PROGRAM Y_Axis
VAR

END_VAR



TrucY();

METHOD TrucY : BOOL
VAR_INPUT
END_VAR
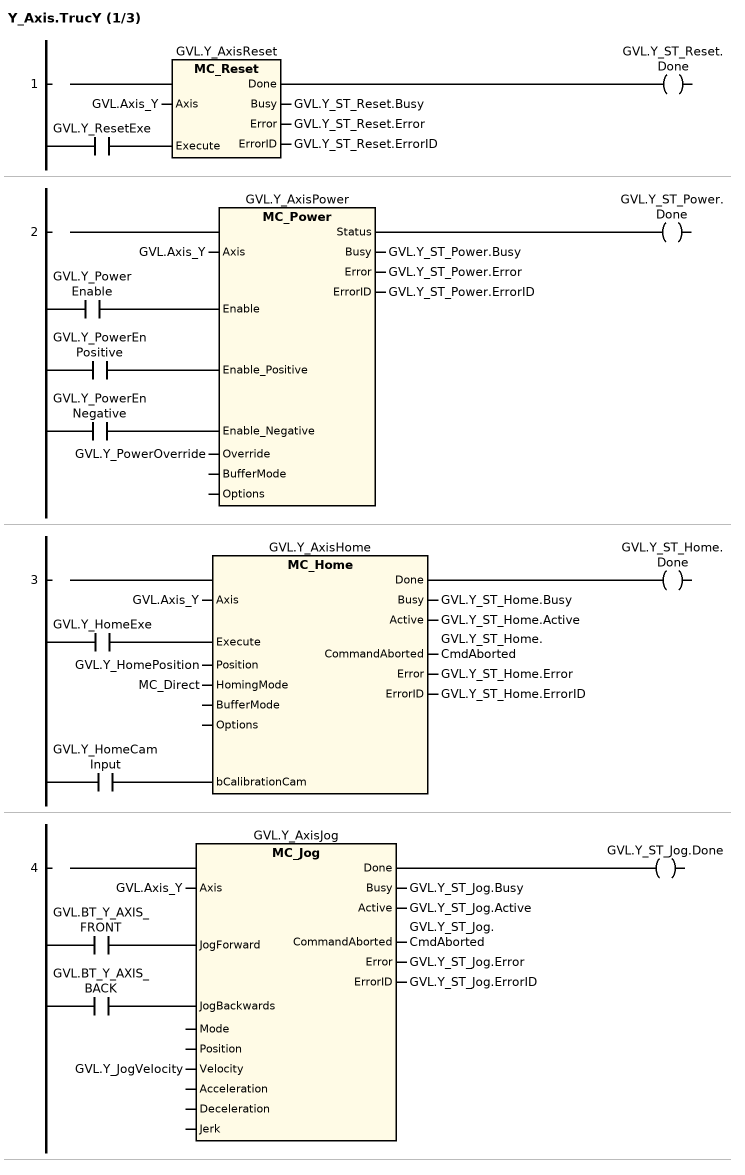
// NETWORK 1
GVL.Y_AxisReset(
    Axis := GVL.Axis_Y,
    Execute := GVL.Y_ResetExe,
    Busy => GVL.Y_ST_Reset.Busy,
    Error => GVL.Y_ST_Reset.Error,
    ErrorID => GVL.Y_ST_Reset.ErrorID); // MC_Reset
GVL.Y_ST_Reset.Done := GVL.Y_AxisReset.Done;

// NETWORK 2
GVL.Y_AxisPower(
    Axis := GVL.Axis_Y,
    Enable := GVL.Y_PowerEnable,
    Enable_Positive := GVL.Y_PowerEnPositive,
    Enable_Negative := GVL.Y_PowerEnNegative,
    Override := GVL.Y_PowerOverride,
    Busy => GVL.Y_ST_Power.Busy,
    Error => GVL.Y_ST_Power.Error,
    ErrorID => GVL.Y_ST_Power.ErrorID); // MC_Power
GVL.Y_ST_Power.Done := GVL.Y_AxisPower.Status;

// NETWORK 3
GVL.Y_AxisHome(
    Axis := GVL.Axis_Y,
    Execute := GVL.Y_HomeExe,
    Position := GVL.Y_HomePosition,
    HomingMode := MC_Direct,
    bCalibrationCam := GVL.Y_HomeCamInput,
    Busy => GVL.Y_ST_Home.Busy,
    Active => GVL.Y_ST_Home.Active,
    CommandAborted => GVL.Y_ST_Home.CmdAborted,
    Error => GVL.Y_ST_Home.Error,
    ErrorID => GVL.Y_ST_Home.ErrorID); // MC_Home
GVL.Y_ST_Home.Done := GVL.Y_AxisHome.Done;

// NETWORK 4
GVL.Y_AxisJog(
    Axis := GVL.Axis_Y,
    JogForward := GVL.BT_Y_AXIS_FRONT,
    JogBackwards := GVL.BT_Y_AXIS_BACK,
    Velocity := GVL.Y_JogVelocity,
    Busy => GVL.Y_ST_Jog.Busy,
    Active => GVL.Y_ST_Jog.Active,
    CommandAborted => GVL.Y_ST_Jog.CmdAborted,
    Error => GVL.Y_ST_Jog.Error,
    ErrorID => GVL.Y_ST_Jog.ErrorID); // MC_Jog
GVL.Y_ST_Jog.Done := GVL.Y_AxisJog.Done;

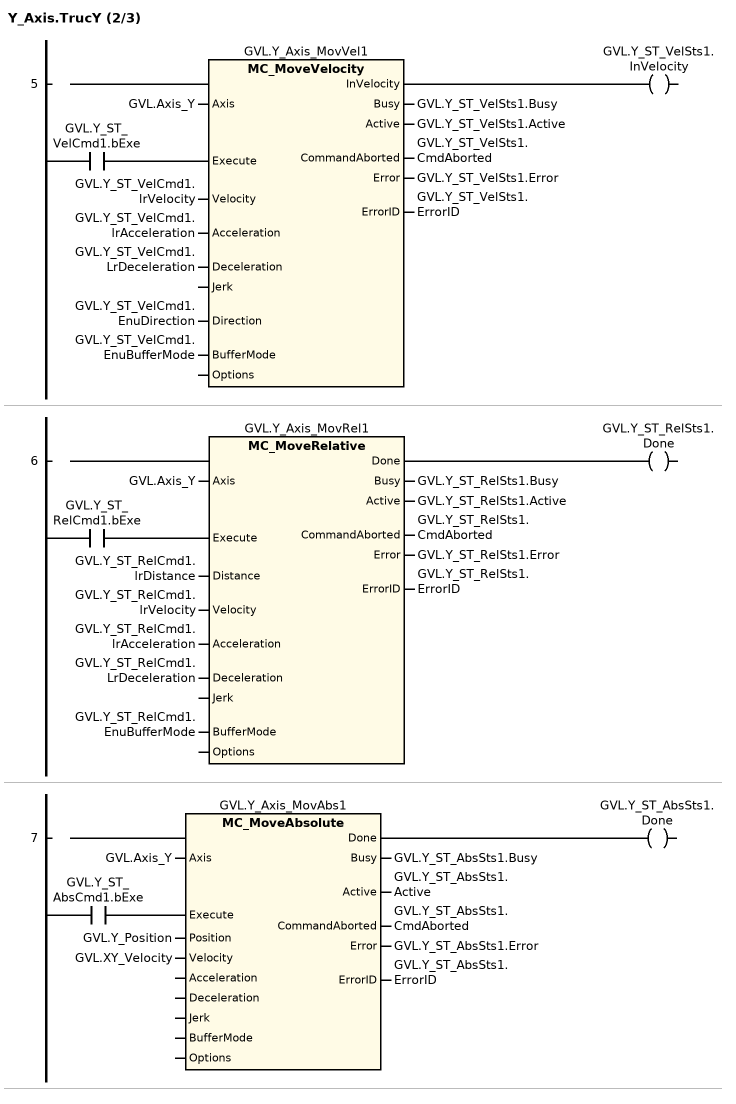
// NETWORK 5
GVL.Y_Axis_MovVel1(
    Axis := GVL.Axis_Y,
    Execute := GVL.Y_ST_VelCmd1.bExe,
    Velocity := GVL.Y_ST_VelCmd1.lrVelocity,
    Acceleration := GVL.Y_ST_VelCmd1.lrAcceleration,
    Deceleration := GVL.Y_ST_VelCmd1.LrDeceleration,
    Direction := GVL.Y_ST_VelCmd1.EnuDirection,
    BufferMode := GVL.Y_ST_VelCmd1.EnuBufferMode,
    Busy => GVL.Y_ST_VelSts1.Busy,
    Active => GVL.Y_ST_VelSts1.Active,
    CommandAborted => GVL.Y_ST_VelSts1.CmdAborted,
    Error => GVL.Y_ST_VelSts1.Error,
    ErrorID => GVL.Y_ST_VelSts1.ErrorID); // MC_MoveVelocity
GVL.Y_ST_VelSts1.InVelocity := GVL.Y_Axis_MovVel1.InVelocity;

// NETWORK 6
GVL.Y_Axis_MovRel1(
    Axis := GVL.Axis_Y,
    Execute := GVL.Y_ST_RelCmd1.bExe,
    Distance := GVL.Y_ST_RelCmd1.lrDistance,
    Velocity := GVL.Y_ST_RelCmd1.lrVelocity,
    Acceleration := GVL.Y_ST_RelCmd1.lrAcceleration,
    Deceleration := GVL.Y_ST_RelCmd1.LrDeceleration,
    BufferMode := GVL.Y_ST_RelCmd1.EnuBufferMode,
    Busy => GVL.Y_ST_RelSts1.Busy,
    Active => GVL.Y_ST_RelSts1.Active,
    CommandAborted => GVL.Y_ST_RelSts1.CmdAborted,
    Error => GVL.Y_ST_RelSts1.Error,
    ErrorID => GVL.Y_ST_RelSts1.ErrorID); // MC_MoveRelative
GVL.Y_ST_RelSts1.Done := GVL.Y_Axis_MovRel1.Done;

// NETWORK 7
GVL.Y_Axis_MovAbs1(
    Axis := GVL.Axis_Y,
    Execute := GVL.Y_ST_AbsCmd1.bExe,
    Position := GVL.Y_Position,
    Velocity := GVL.XY_Velocity,
    Busy => GVL.Y_ST_AbsSts1.Busy,
    Active => GVL.Y_ST_AbsSts1.Active,
    CommandAborted => GVL.Y_ST_AbsSts1.CmdAborted,
    Error => GVL.Y_ST_AbsSts1.Error,
    ErrorID => GVL.Y_ST_AbsSts1.ErrorID); // MC_MoveAbsolute
GVL.Y_ST_AbsSts1.Done := GVL.Y_Axis_MovAbs1.Done;

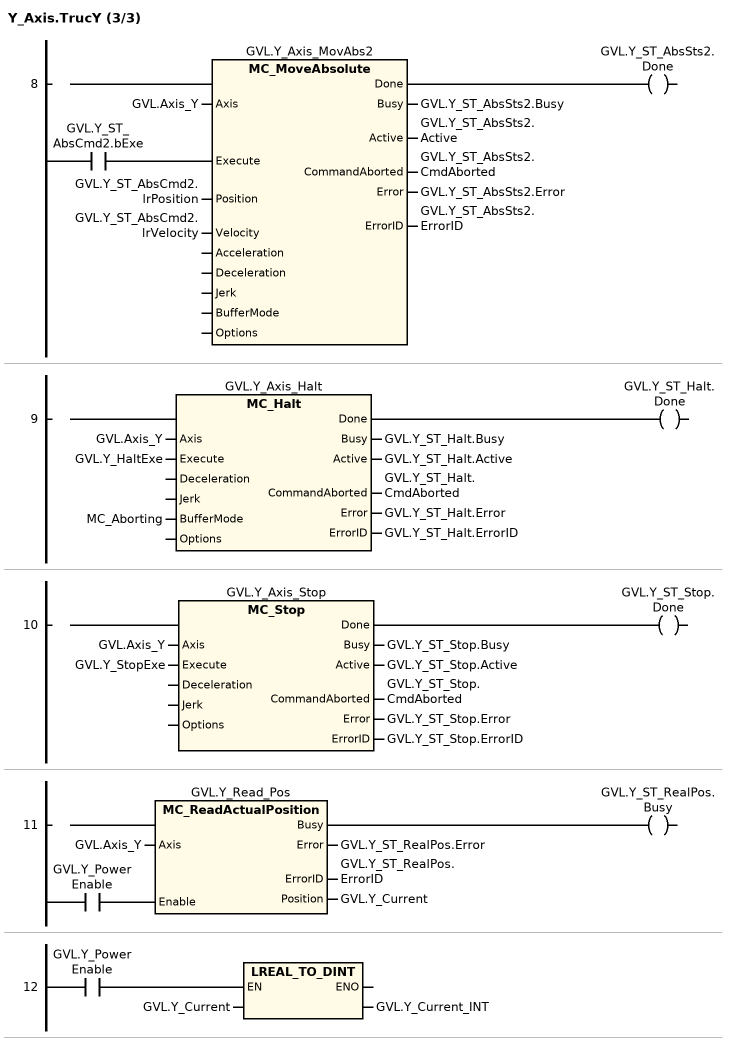
// NETWORK 8
GVL.Y_Axis_MovAbs2(
    Axis := GVL.Axis_Y,
    Execute := GVL.Y_ST_AbsCmd2.bExe,
    Position := GVL.Y_ST_AbsCmd2.lrPosition,
    Velocity := GVL.Y_ST_AbsCmd2.lrVelocity,
    Busy => GVL.Y_ST_AbsSts2.Busy,
    Active => GVL.Y_ST_AbsSts2.Active,
    CommandAborted => GVL.Y_ST_AbsSts2.CmdAborted,
    Error => GVL.Y_ST_AbsSts2.Error,
    ErrorID => GVL.Y_ST_AbsSts2.ErrorID); // MC_MoveAbsolute
GVL.Y_ST_AbsSts2.Done := GVL.Y_Axis_MovAbs2.Done;

// NETWORK 9
GVL.Y_Axis_Halt(
    Axis := GVL.Axis_Y,
    Execute := GVL.Y_HaltExe,
    BufferMode := MC_Aborting,
    Busy => GVL.Y_ST_Halt.Busy,
    Active => GVL.Y_ST_Halt.Active,
    CommandAborted => GVL.Y_ST_Halt.CmdAborted,
    Error => GVL.Y_ST_Halt.Error,
    ErrorID => GVL.Y_ST_Halt.ErrorID); // MC_Halt
GVL.Y_ST_Halt.Done := GVL.Y_Axis_Halt.Done;

// NETWORK 10
GVL.Y_Axis_Stop(
    Axis := GVL.Axis_Y,
    Execute := GVL.Y_StopExe,
    Busy => GVL.Y_ST_Stop.Busy,
    Active => GVL.Y_ST_Stop.Active,
    CommandAborted => GVL.Y_ST_Stop.CmdAborted,
    Error => GVL.Y_ST_Stop.Error,
    ErrorID => GVL.Y_ST_Stop.ErrorID); // MC_Stop
GVL.Y_ST_Stop.Done := GVL.Y_Axis_Stop.Done;

// NETWORK 11
GVL.Y_Read_Pos(
    Axis := GVL.Axis_Y,
    Enable := GVL.Y_PowerEnable,
    Busy => GVL.Y_ST_RealPos.Busy,
    Error => GVL.Y_ST_RealPos.Error,
    ErrorID => GVL.Y_ST_RealPos.ErrorID,
    Position => GVL.Y_Current); // MC_ReadActualPosition

// NETWORK 12
IF GVL.Y_PowerEnable THEN GVL.Y_Current_INT := LREAL_TO_DINT(GVL.Y_Current); END_IF
END_METHOD

END_PROGRAM

(* stored: Version 1.1.0.1, ProductVersion 3.1.4024.13
   POU Y_Axis: Id {550eefd2-e8b6-4fc6-bcf2-ab345ba4d8a4}, SpecialFunc None
   Method TrucY: Id {b0e69374-00cd-485c-9d7d-2f76380d4f74} *)
